Staubli VAL3: screenUpdate.pgx

public program screenUpdate()
  local num l_nExecStatus
  local num l_nElems
begin
  // Copyright (c) 2016, Ocado Technology - Robotics Research Team
  //
  // Licensed under the Apache License, Version 2.0 (the "License");
  // you may not use this file except in compliance with the License.
  // You may obtain a copy of the License at
  //
  //     http://www.apache.org/licenses/LICENSE-2.0
  //
  // Unless required by applicable law or agreed to in writing, software
  // distributed under the License is distributed on an "AS IS" BASIS,
  // WITHOUT WARRANTIES OR CONDITIONS OF ANY KIND, either express or implied.
  // See the License for the specific language governing permissions and
  // limitations under the License.

  l_nExecStatus = 0

  call libInterface:init()

  while(true)

    // clear screen
    call libInterface:clearScreen()

    // update connection status on port 11000
    call libInterface:motionStatus(nInConnFlag)

    // update connection status on port 11002
    call libInterface:feedbackStatus(nOutConnFlag)

    // update trajectory buffer size
    call libQueueFuncs:getNumElems(qTrajPtBuffer,l_nElems)
    call libInterface:trajBuffer(l_nElems,nPtsPopped)

    // do the same for move buffer
    call libQueueFuncs:getNumElems(qMoveBuffer,l_nElems)
    call libInterface:motionBuffer(l_nElems,nPtsPopped)

    // display nMoveId and nMotionProgress
    call libInterface:motionProgress(nMoveId,nMotionProgress)

    // display time between valid trajectory point received and ACK sent
    call libInterface:ack(nHeaderTime,nElapsedTime)

    // update debug status
    call libInterface:debug(l_nExecStatus)

    //    // add Function keys labels
    //    gotoxy(scMonitor, 30,13)
    //    put(scMonitor, "V/ON")
    //    gotoxy(scMonitor, 35,13)
    //    put(scMonitor, "V/OFF")

    // sequence task
    //delay(0)
    delay(0.5)
  endWhile
end
